Fanuc KAREL source: kx00001.KL

-- PROVISIONAL review KL for V1013-1; original PC SHA256 86eac0b3f2daa2e0d35417fbfe8b5a5de8c511fa2a34b95cd63fe1b66203effa
-- Incomplete behavior may be omitted. Consult companion uncertainty JSON. Do not deploy.
PROGRAM KX00001
%NOLOCKGROUP
VAR
  I : INTEGER
  J : INTEGER
  B : BOOLEAN
  F : FILE
  S : STRING[80]
-- UNRESOLVED_DECL P type=000102
BEGIN
  -- UNRESOLVED_PC offsets 5-32; opcodes 22,3F,3F,3D
  -- UNRESOLVED_PC offsets 37-41; opcodes 7F
END KX00001
